PROGRAM MAIN
VAR
END_VAR

F_ConsumeTime(75);

END_PROGRAM

(* stored: Version 1.1.0.1, ProductVersion 3.1.4026.18
   POU MAIN: Id {c98c3423-108a-4149-8932-7c95b5e5cea3}, SpecialFunc None *)
